{attribute 'c++_compatible'}
FUNCTION_BLOCK FB_MyMqtt EXTENDS FB_IotMqttClient
VAR_INPUT
END_VAR
VAR_OUTPUT
END_VAR
VAR
	(* received message *)
    {attribute 'TcEncoding':='UTF-8'}
    sTopicRcv   : STRING(255);
    {attribute 'TcEncoding':='UTF-8'}
    sPayloadRcv : STRING(255);
END_VAR

{attribute 'c++_compatible'}
{attribute 'pack_mode' := '4'}
{attribute 'show'}
{attribute 'minimal_input_size' := '4'}
METHOD OnMqttMessage : HRESULT
VAR_IN_OUT CONSTANT
    topic    : STRING;
END_VAR
VAR_INPUT
    payload  : PVOID;
    length   : UDINT;
    qos      : TcIotMqttQos;
    repeated : BOOL;
END_VAR
VAR
    nPayloadRcvLen : UDINT;
END_VAR
SUPER^.nMessagesRcv := SUPER^.nMessagesRcv + 1;

STRNCPY( ADR(sTopicRcv), ADR(topic), SIZEOF(sTopicRcv) );
nPayloadRcvLen := MIN(length, DINT_TO_UDINT(SIZEOF(sPayloadRcv))-1);
MEMCPY( ADR(sPayloadRcv), payload, nPayloadRcvLen );
sPayloadRcv[nPayloadRcvLen] := 0;  // ensure a null termination of received string

OnMqttMessage := S_OK;
END_METHOD

END_FUNCTION_BLOCK

(* stored: Version 1.1.0.1, ProductVersion 3.1.4024.15
   POU FB_MyMqtt: Id {933e564c-2550-4fc2-a337-abe6d6bb0cff}, SpecialFunc None
   Method OnMqttMessage: Id {cc89d025-68ae-4893-a436-356ed18f84b6} *)
